INTERFACE I_SafetySimulation EXTENDS I_Simulatable

METHOD SimulateSafetyDiag
VAR_INPUT
	SimulationValueDiag : UINT;
END_VAR
END_METHOD

METHOD SimulateSafetyState
VAR_INPUT
	SimulationValueState : USINT;
END_VAR
END_METHOD

END_INTERFACE

(* stored: Version 1.1.0.1, ProductVersion 3.1.4026.18
   Itf I_SafetySimulation: Id {ca0cee81-6bde-08e0-02c6-6f5bea10c344}
   Method SimulateSafetyDiag: Id {e9ca0188-4ac0-4a84-8ea6-cb92241a0d24}
   Method SimulateSafetyState: Id {bc0695d1-1e1a-4e72-bf9c-768eb9226d50} *)
